// TIA Portal V16 export
// export: Created 2022-11-17T15:49:45.0042445Z, ExportSetting WithDefaults, DisplayName Totally Integrated Automation Portal, DisplayVersion V16 Update 6, DisplayName TIA Portal Version Control Interface, DisplayVersion V16 Update 2, DisplayName TIA Portal Openness, DisplayVersion V16 Update 6, DisplayName SINAMICS Startdrive Advanced, DisplayVersion V16 Update 5, DisplayName SINAMICS Startdrive G130, G150, S120, S150, SINAMICS MV, S210, DisplayVersion V16 Update 5, DisplayName SINAMICS Startdrive G110M, G120, G120C, G120D, G120P, G115D, DisplayVersion V16 Update 5, DisplayName STEP 7 Professional, DisplayVersion V16 Update 6, DisplayName STEP 7 Safety, DisplayVersion V16, DisplayName WinCC Advanced, DisplayVersion V16 Update 6
DATA_BLOCK "DB243_Program7"   // DB243
{ S7_Optimized_Access := 'FALSE' }
AUTHOR : Robopac
VERSION : 0.0
// stored: AutoNumber false, IsOnlyStoredInLoadMemory false, IsWriteProtectedInAS false
   VAR RETAIN
      Program7 { S7_SetPoint := 'True'} : "DatiProgramma";
   END_VAR
BEGIN
   Program7.Wrapping := TRUE;
   Program7.TopLenght := 500;
   Program7.TopRelease := 0;
   Program7.TopDown := 0;
   Program7.Top := 4;
   Program7.PressurePTime := 0;
   Program7.LifterTime := 0;
   Program7.RevOverContrast := 1;
   Program7.RopeEndCycle := 16#01;
   Program7.Spare4 := 16#01;
   Program7.RopeTime := 1500;
   Program7.RevOverClamp := 1;
   Program7.FilmForceFinalRev := 15;
   Program7.FilmPrestretchFinalRev := 100;
   Program7.ArmSpeed := 100;
   Program7.CarriageDown4Top := 500;
   Program7.TopDownTime := 1500;
   Program7.LapsUnderTop := 0;
   Program7.Spare6 := 0;
   Program7.Spare7 := 0;
   Program7.Spare8 := 0;
   Program7.Spare9 := 0;
   Program7.Spare10 := 0;
   Program7.Spare11 := 0;
   Program7.Spare12 := 0;
   Program7.Overlap0_1 := 0;
   Program7.Height1 := 15;
   Program7.Landmark1 := FALSE;
   Program7.Lifter1 := FALSE;
   Program7.SpareBit1H1 := FALSE;
   Program7.Airblower1 := TRUE;
   Program7.NextStep1 := TRUE;
   Program7.PressureP1 := TRUE;
   Program7.SpareByte2H1 := 16#00;
   Program7.Revolution1 := 0;
   Program7.RopeUnit1_1 := 16#02;
   Program7.RopeUnit1_2 := 16#01;
   Program7.FilmForce1 := 5;
   Program7.FilmPrestretch1 := 200;
   Program7.Spare3H1 := 0;
   Program7.Spare49 := 0;
   Program7.Spare50 := 0;
   Program7.Spare51 := 0;
   Program7.Spare52 := 0;
   Program7.Spare53 := 0;
   Program7.Overlap1_2 := 0;
   Program7.Height2 := 80;
   Program7.Landmark2 := FALSE;
   Program7.Lifter2 := FALSE;
   Program7.SpareBit1H2 := FALSE;
   Program7.Airblower2 := TRUE;
   Program7.NextStep2 := TRUE;
   Program7.PressureP2 := TRUE;
   Program7.SpareByte2H2 := 16#00;
   Program7.Revolution2 := 1;
   Program7.RopeUnit2_1 := 16#01;
   Program7.RopeUnit2_2 := 16#01;
   Program7.FilmForce2 := 15;
   Program7.FilmPrestretch2 := 200;
   Program7.Spare3H2 := 0;
   Program7.Spare54 := 0;
   Program7.Spare55 := 0;
   Program7.Spare56 := 0;
   Program7.Spare57 := 0;
   Program7.Spare58 := 0;
   Program7.Overlap2_3 := 0;
   Program7.Height3 := 120;
   Program7.Landmark3 := FALSE;
   Program7.Lifter3 := FALSE;
   Program7.SpareBit1H3 := FALSE;
   Program7.Airblower3 := TRUE;
   Program7.NextStep3 := TRUE;
   Program7.PressureP3 := TRUE;
   Program7.SpareByte2H3 := 16#00;
   Program7.Revolution3 := 1;
   Program7.RopeUnit3_1 := 16#01;
   Program7.RopeUnit3_2 := 16#01;
   Program7.FilmForce3 := 25;
   Program7.FilmPrestretch3 := 200;
   Program7.Spare3H3 := 0;
   Program7.Spare59 := 0;
   Program7.Spare60 := 0;
   Program7.Spare61 := 380;
   Program7.Spare62 := 2800;
   Program7.Spare63 := 0;
   Program7.Overlap3_4 := 0;
   Program7.Height4 := -100;
   Program7.Landmark4 := TRUE;
   Program7.Lifter4 := FALSE;
   Program7.SpareBit1H4 := FALSE;
   Program7.Airblower4 := FALSE;
   Program7.NextStep4 := TRUE;
   Program7.PressureP4 := TRUE;
   Program7.SpareByte2H4 := 16#00;
   Program7.Revolution4 := 1;
   Program7.RopeUnit4_1 := 16#01;
   Program7.RopeUnit4_2 := 16#01;
   Program7.FilmForce4 := 20;
   Program7.FilmPrestretch4 := 200;
   Program7.Spare3H4 := 0;
   Program7.Spare64 := 0;
   Program7.Spare65 := 0;
   Program7.Spare66 := 0;
   Program7.Spare67 := 0;
   Program7.Spare68 := 0;
   Program7.Overlap4_5 := 300;
   Program7.Height5 := 120;
   Program7.Landmark5 := FALSE;
   Program7.Lifter5 := FALSE;
   Program7.SpareBit1H5 := FALSE;
   Program7.Airblower5 := TRUE;
   Program7.NextStep5 := TRUE;
   Program7.PressureP5 := FALSE;
   Program7.SpareByte2H5 := 16#00;
   Program7.Revolution5 := 2;
   Program7.RopeUnit5_1 := 16#02;
   Program7.RopeUnit5_2 := 16#02;
   Program7.FilmForce5 := 15;
   Program7.FilmPrestretch5 := 200;
   Program7.Spare3H5 := 0;
   Program7.Spare69 := 0;
   Program7.Spare70 := 0;
   Program7.Spare71 := 0;
   Program7.Spare72 := 0;
   Program7.Spare73 := 0;
   Program7.Overlap5_6 := 300;
   Program7.Height6 := 85;
   Program7.Landmark6 := FALSE;
   Program7.Lifter6 := FALSE;
   Program7.SpareBit1H6 := FALSE;
   Program7.Airblower6 := TRUE;
   Program7.NextStep6 := FALSE;
   Program7.PressureP6 := FALSE;
   Program7.SpareByte2H6 := 16#00;
   Program7.Revolution6 := 1;
   Program7.RopeUnit6_1 := 16#01;
   Program7.RopeUnit6_2 := 16#01;
   Program7.FilmForce6 := 20;
   Program7.FilmPrestretch6 := 200;
   Program7.Spare3H6 := 0;
   Program7.Spare74 := 0;
   Program7.Spare75 := 0;
   Program7.Spare76 := 0;
   Program7.Spare77 := 0;
   Program7.Spare78 := 0;
   Program7.Overlap6_7 := 0;
   Program7.Height7 := 0;
   Program7.Landmark7 := FALSE;
   Program7.Lifter7 := FALSE;
   Program7.SpareBit1H7 := FALSE;
   Program7.Airblower7 := FALSE;
   Program7.NextStep7 := TRUE;
   Program7.PressureP7 := FALSE;
   Program7.SpareByte2H7 := 16#00;
   Program7.Revolution7 := 1;
   Program7.RopeUnit7_1 := 16#01;
   Program7.RopeUnit7_2 := 16#01;
   Program7.FilmForce7 := 0;
   Program7.FilmPrestretch7 := 100;
   Program7.Spare3H7 := 0;
   Program7.Spare79 := 0;
   Program7.Spare80 := 0;
   Program7.Spare81 := 0;
   Program7.Spare82 := 0;
   Program7.Spare83 := 0;
   Program7.Overlap7_8 := 0;
   Program7.Height8 := 0;
   Program7.Landmark8 := FALSE;
   Program7.Lifter8 := FALSE;
   Program7.SpareBit1H8 := FALSE;
   Program7.Airblower8 := FALSE;
   Program7.NextStep8 := TRUE;
   Program7.PressureP8 := FALSE;
   Program7.SpareByte2H8 := 16#00;
   Program7.Revolution8 := 1;
   Program7.RopeUnit8_1 := 16#01;
   Program7.RopeUnit8_2 := 16#01;
   Program7.FilmForce8 := 0;
   Program7.FilmPrestretch8 := 100;
   Program7.Spare3H8 := 0;
   Program7.Spare84 := 0;
   Program7.Spare85 := 0;
   Program7.Spare86 := 0;
   Program7.Spare87 := 0;
   Program7.Spare88 := 0;
   Program7.Overlap8_9 := 0;
   Program7.Height9 := 0;
   Program7.Landmark9 := FALSE;
   Program7.Lifter9 := FALSE;
   Program7.SpareBit1H9 := FALSE;
   Program7.Airblower9 := FALSE;
   Program7.NextStep9 := TRUE;
   Program7.PressureP9 := FALSE;
   Program7.SpareByte2H9 := 16#00;
   Program7.Revolution9 := 1;
   Program7.RopeUnit9_1 := 16#01;
   Program7.RopeUnit9_2 := 16#01;
   Program7.FilmForce9 := 0;
   Program7.FilmPrestretch9 := 100;
   Program7.Spare3H9 := 0;
   Program7.Spare89 := 0;
   Program7.Spare90 := 0;
   Program7.Spare91 := 0;
   Program7.Spare92 := 0;
   Program7.Spare93 := 0;
   Program7.Overlap9_10 := 0;
   Program7.Height10 := 0;
   Program7.Landmark10 := FALSE;
   Program7.Lifter10 := FALSE;
   Program7.SpareBit1H10 := FALSE;
   Program7.Airblower10 := FALSE;
   Program7.NextStep10 := FALSE;
   Program7.PressureP10 := FALSE;
   Program7.SpareByte2H10 := 16#00;
   Program7.Revolution10 := 1;
   Program7.RopeUnit10_1 := 16#01;
   Program7.RopeUnit10_2 := 16#01;
   Program7.FilmForce10 := 0;
   Program7.FilmPrestretch10 := 100;
   Program7.Spare3H10 := 0;
   Program7.Spare94 := 0;
   Program7.Spare95 := 0;
   Program7.Spare96 := 0;
   Program7.Spare97 := 0;
   Program7.Spare98 := 0;
   Program7.Overlap10_11 := 0;
   Program7.Height11 := 0;
   Program7.Landmark11 := FALSE;
   Program7.Lifter11 := FALSE;
   Program7.SpareBit1H11 := FALSE;
   Program7.Airblower11 := FALSE;
   Program7.NextStep11 := TRUE;
   Program7.PressureP11 := FALSE;
   Program7.SpareByte2H11 := 16#00;
   Program7.Revolution11 := 1;
   Program7.RopeUnit11_1 := 16#01;
   Program7.RopeUnit11_2 := 16#01;
   Program7.FilmForce11 := 0;
   Program7.FilmPrestretch11 := 100;
   Program7.Spare3H11 := 0;
   Program7.Spare99 := 0;
   Program7.Spare100 := 0;
   Program7.Spare101 := 0;
   Program7.Spare102 := 0;
   Program7.Spare103 := 0;
   Program7.Overlap11_12 := 0;
   Program7.Height12 := 0;
   Program7.Landmark12 := FALSE;
   Program7.Lifter12 := FALSE;
   Program7.SpareBit1H12 := FALSE;
   Program7.Airblower12 := FALSE;
   Program7.NextStep12 := FALSE;
   Program7.PressureP12 := FALSE;
   Program7.SpareByte2H12 := 16#00;
   Program7.Revolution12 := 1;
   Program7.RopeUnit12_1 := 16#01;
   Program7.RopeUnit12_2 := 16#01;
   Program7.FilmForce12 := 0;
   Program7.FilmPrestretch12 := 100;
   Program7.Spare3H12 := 0;
   Program7.Spare104 := 0;
   Program7.Spare105 := 0;
   Program7.Spare106 := 0;
   Program7.Spare107 := 0;
   Program7.Spare108 := 0;
END_DATA_BLOCK
